(* IEC 61131-3 sources: std_i2980_v2.06_cp053/Source/IMM/ieccontrol/Scope (part 2) *)

(* ---- ABScopeTrigger.pu ---- *)
(*
@h    ! WARNING !
@h    The Kemro K2 system (including software) only meets category B according to EN 954-1,
@h    thus it is not intended for usage in safety-relevant control applications in the field
@h    of personal safety (e.g. emergency stop).
@h    To implement potentially necessary safety-relevant control tasks, always use additional
@h    external safety devices that are intended for the particular purpose, and meet the necessary
@h    functional safety.
@h    For further information see EN 954-1 (EN ISO 13849-1) and/or the K2-x00 user manual, chapter
@h    "CE conformity, directives and standards".

*)

IMPORT_OVER_LISTFILE
 START_PROCESS_ALGORITHM
, cCompMold
, cMoveFwdInterPos
, cMoveFwd
, cMoveBwd
, cMoveBwdInterPos
, cCompInjection
, cMoveInject
, cMovePlast
, TON
, tevMovementState
, tpTriggerData
, tsTriggerData
, tevMovementStateData
, tnActiveInactive

END_IMPORT

ALGORITHM_BLOCK ABScopeTrigger #DUMMY_EDIT_BLOCK

SYSTEM_OBJECT
 PU_Task_7 : TASK;
 EV_Task_3 : TASK;
 Task10ms : TASK;
 evMovementState : tevMovementState;
END_OBJECT

VAR
 fbTimer : TON;
 mevMovementState : tevMovementState (* movement state event *);
 mpbCustomVarTriggerPU : REFTO BOOL;
 mpTriggerPU : tpTriggerData;
 mpTrigger : tpTriggerData;
 mbInit : BOOL;
END_VAR

ALGORITHM aReset

#BEGIN_EDIT_BLOCK
(**************************************** WARNING ********************************************
 *** The KEBA Kemro K2 System including software is not intended for safety control tasks! ***
 ***                       For further information see Comment tab!                        ***
 *********************************************************************************************)

IF (NOT mbInit) THEN
   RETURN;
END_IF;

mpTrigger^.iState := 0;
mpTrigger^.Reduction.iAct := 0;

;#END_EDIT_BLOCK END_ALGORITHM

FUNCTION fArm : BOOL
 #DUMMY_EDIT_BLOCK

VAR_INPUT
 bArm : BOOL (* true activates the waiting for the trigger event *);
END_VAR
#BEGIN_EDIT_BLOCK
(**************************************** WARNING ********************************************
 *** The KEBA Kemro K2 System including software is not intended for safety control tasks! ***
 ***                       For further information see Comment tab!                        ***
 *********************************************************************************************)

IF (NOT mbInit) THEN
   RETURN;
END_IF;

mpTrigger^.bTriggered := FALSE;
mpTrigger^.bPreTriggered := FALSE;
mevMovementState := EMPTY;
mpbCustomVarTriggerPU := EMPTY;
mpTriggerPU := EMPTY;

STOP_PROCESS_ALGORITHM(paTriggerDelay);

IF bArm THEN
   // activate the events
   CASE mpTrigger^.iTriggerIdx OF
      0: // no trigger
         RETURN;

      1..4: // movement triggers
         mevMovementState := evMovementState;

      5: // variable trigger
         mpTrigger^.pbCustomVarTrigger^ := FALSE;
         mpbCustomVarTriggerPU := mpTrigger^.pbCustomVarTrigger;

   END_CASE;
   mpTriggerPU := mpTrigger;
   mpTrigger^.Reduction.iAct := 0;
   mpTrigger^.iState := 1;
END_IF;

fArm := TRUE;

;#END_EDIT_BLOCK END_FUNCTION

FUNCTION fCheckMovementTrigger : BOOL
 #DUMMY_EDIT_BLOCK

VAR_INPUT
 triggerData : tsTriggerData;
 evMovementStateData : tevMovementStateData;
END_VAR

VAR
 nState : tnActiveInactive;
END_VAR
#BEGIN_EDIT_BLOCK
(**************************************** WARNING ********************************************
 *** The KEBA Kemro K2 System including software is not intended for safety control tasks! ***
 ***                       For further information see Comment tab!                        ***
 *********************************************************************************************)

fCheckMovementTrigger := FALSE;

nState := nActive;
IF (triggerData.bFallingEdge) THEN
   nState := nInactive;
END_IF;

IF (evMovementStateData.State = nState) AND
   (//mold close (interposition)
   (triggerData.iTriggerIdx = 1 AND evMovementStateData.DeviceId.CompId = cCompMold AND
   evMovementStateData.DeviceId.IndexId = 1 AND (evMovementStateData.MoveId = cMoveFwdInterPos OR evMovementStateData.MoveId = cMoveFwd) AND
   evMovementStateData.MoveDir = cMoveFwd) OR
   //mold open (interposition)
   (triggerData.iTriggerIdx = 2 AND evMovementStateData.DeviceId.CompId = cCompMold AND
   evMovementStateData.DeviceId.IndexId = 1 AND (evMovementStateData.MoveId = cMoveBwdInterPos OR evMovementStateData.MoveId = cMoveBwd) AND
   evMovementStateData.MoveDir = cMoveBwd) OR
   //inject
   (triggerData.iTriggerIdx = 3 AND evMovementStateData.DeviceId.CompId = cCompInjection AND
   evMovementStateData.DeviceId.IndexId = 1 AND evMovementStateData.MoveId = cMoveInject AND
   evMovementStateData.MoveDir = cMoveFwd) OR
   //plast
   (triggerData.iTriggerIdx = 4 AND evMovementStateData.DeviceId.CompId = cCompInjection AND
   evMovementStateData.DeviceId.IndexId = 1 AND evMovementStateData.MoveId = cMovePlast AND
   evMovementStateData.MoveDir = cMoveBwd)) THEN

   fCheckMovementTrigger := TRUE;
END_IF;

;#END_EDIT_BLOCK END_FUNCTION

ALGORITHM aTrigger

#BEGIN_EDIT_BLOCK
(**************************************** WARNING ********************************************
 *** The KEBA Kemro K2 System including software is not intended for safety control tasks! ***
 ***                       For further information see Comment tab!                        ***
 *********************************************************************************************)

// after ingnition occured, trigger immediately or wait until delay expired
IF (mpTrigger^.dTriggerDelay > t#0.0s) THEN
   fbTimer(IN := FALSE);
   START_PROCESS_ALGORITHM(paTriggerDelay);
ELSE
   // trigger immediately
   mpTrigger^.bTriggered := TRUE;
   mpTrigger^.iState := 2;
END_IF;

;#END_EDIT_BLOCK END_ALGORITHM

ALGORITHM aInit

VAR_INPUT
 pTrigger : tpTriggerData;
END_VAR

VAR
 b : BOOL;
END_VAR
#BEGIN_EDIT_BLOCK
(**************************************** WARNING ********************************************
 *** The KEBA Kemro K2 System including software is not intended for safety control tasks! ***
 ***                       For further information see Comment tab!                        ***
 *********************************************************************************************)

mpTrigger := pTrigger;
mpTriggerPU := EMPTY;
mpbCustomVarTriggerPU := EMPTY;

fbTimer(IN := FALSE);

b := fArm(FALSE);
aReset();

mbInit := TRUE;

;#END_EDIT_BLOCK END_ALGORITHM

PROCESS_ALGORITHM paTriggerDelay ON Task10ms

#BEGIN_EDIT_BLOCK
(**************************************** WARNING ********************************************
 *** The KEBA Kemro K2 System including software is not intended for safety control tasks! ***
 ***                       For further information see Comment tab!                        ***
 *********************************************************************************************)

fbTimer(IN := TRUE, PT := mpTrigger^.dTriggerDelay);

IF fbTimer.Q THEN
   // time-trigger after trigger is ignited and delay is expired
   mpTrigger^.bTriggered := TRUE;
   mpTrigger^.iState := 2;
   STOP_PROCESS_ALGORITHM();
END_IF;

;#END_EDIT_BLOCK END_ALGORITHM

POSTUPDATE_ALGORITHM pPreTriggered ON PU_Task_7 WITH mpTriggerPU^.bPreTriggered

#BEGIN_EDIT_BLOCK
(**************************************** WARNING ********************************************
 *** The KEBA Kemro K2 System including software is not intended for safety control tasks! ***
 ***                       For further information see Comment tab!                        ***
 *********************************************************************************************)

IF (NOT mbInit) THEN
   RETURN;
END_IF;

IF (mpTrigger^.bPreTriggered AND mpTrigger^.Reduction.iAct < mpTrigger^.Reduction.iSet) THEN

   mpTrigger^.Reduction.iAct := mpTrigger^.Reduction.iAct + 1;
   IF (mpTrigger^.Reduction.iAct = mpTrigger^.Reduction.iSet) THEN
      aTrigger();
   END_IF;
   mpTrigger^.bPreTriggered := FALSE;
END_IF;

;#END_EDIT_BLOCK END_ALGORITHM

POSTUPDATE_ALGORITHM pVarTriggered ON PU_Task_7 WITH mpbCustomVarTriggerPU^

#BEGIN_EDIT_BLOCK
(**************************************** WARNING ********************************************
 *** The KEBA Kemro K2 System including software is not intended for safety control tasks! ***
 ***                       For further information see Comment tab!                        ***
 *********************************************************************************************)

IF (mpTrigger^.iTriggerIdx = 5) THEN
   IF ((mpbCustomVarTriggerPU^ AND NOT mpTrigger^.bFallingEdge) OR
       (NOT mpbCustomVarTriggerPU^ AND mpTrigger^.bFallingEdge)) THEN
      mpTrigger^.bPreTriggered := TRUE;
   END_IF;
END_IF;

;#END_EDIT_BLOCK END_ALGORITHM

EVENT_ALGORITHM evaMovementState ON EV_Task_3 WITH mevMovementState

VAR_INPUT
 evMovementStateData : tevMovementStateData;
END_VAR
#BEGIN_EDIT_BLOCK
(**************************************** WARNING ********************************************
 *** The KEBA Kemro K2 System including software is not intended for safety control tasks! ***
 ***                       For further information see Comment tab!                        ***
 *********************************************************************************************)

IF fCheckMovementTrigger(mpTrigger^, evMovementStateData) THEN
   mpTrigger^.bPreTriggered := TRUE;
END_IF;

;#END_EDIT_BLOCK END_ALGORITHM

END_ALGORITHM_BLOCK

#END_OF_IEC_PART

@Puma @IecEditor 6 150 @Pou 25
@@@BEG_Comment@@@
@h    ! WARNING !
@h    The Kemro K2 system (including software) only meets category B according to EN 954-1,
@h    thus it is not intended for usage in safety-relevant control applications in the field
@h    of personal safety (e.g. emergency stop).
@h    To implement potentially necessary safety-relevant control tasks, always use additional
@h    external safety devices that are intended for the particular purpose, and meet the necessary
@h    functional safety.
@h    For further information see EN 954-1 (EN ISO 13849-1) and/or the K2-x00 user manual, chapter
@h    "CE conformity, directives and standards".

@@@END_Comment@@@

@BEG_Contents

@BEG_Func
@RT(17)FuncTreeContainer
1
@Var @RT(23)START_PROCESS_ALGORITHM @RT(0) @T @T @DERIVED 0 @F @RT(23)KEBA_STANDARD_PROCEDURE @F
@T
@BEG_Attrib
0 @RT(0) @RT(0)
@END_Attrib
1 1 @F @F @F @F

@END_Func

@BEG_Const
@RT(18)ConstTreeContainer
8
@Var @RT(9)cCompMold @RT(0) @T @F @DT @RT(4)DINT @RT(0) @T @T @BASIC 0 @F
@F @F
@T
@BEG_Attrib
0 @RT(3)101 @RT(14)Component Mold
@END_Attrib
1 1 @F @F @F @F

@Var @RT(16)cMoveFwdInterPos @RT(0) @T @F @DT @RT(4)DINT @RT(0) @T @T @BASIC 0 @F
@F @F
@T
@BEG_Attrib
0 @RT(2)17 @RT(37)move forward to intermediate position
@END_Attrib
1 1 @F @F @F @F

@Var @RT(8)cMoveFwd @RT(0) @T @F @DT @RT(4)DINT @RT(0) @T @T @BASIC 0 @F
@F @F
@T
@BEG_Attrib
0 @RT(2)12 @RT(16)movement forward
@END_Attrib
1 1 @F @F @F @F

@Var @RT(8)cMoveBwd @RT(0) @T @F @DT @RT(4)DINT @RT(0) @T @T @BASIC 0 @F
@F @F
@T
@BEG_Attrib
0 @RT(2)11 @RT(17)movement backward
@END_Attrib
1 1 @F @F @F @F

@Var @RT(16)cMoveBwdInterPos @RT(0) @T @F @DT @RT(4)DINT @RT(0) @T @T @BASIC 0 @F
@F @F
@T
@BEG_Attrib
0 @RT(2)16 @RT(38)move backward to intermediate position
@END_Attrib
1 1 @F @F @F @F

@Var @RT(14)cCompInjection @RT(0) @T @F @DT @RT(4)DINT @RT(0) @T @T @BASIC 0 @F
@F @F
@T
@BEG_Attrib
0 @RT(3)104 @RT(19)Component Injection
@END_Attrib
1 1 @F @F @F @F

@Var @RT(11)cMoveInject @RT(0) @T @F @DT @RT(4)DINT @RT(0) @T @T @BASIC 0 @F
@F @F
@T
@BEG_Attrib
0 @RT(2)14 @RT(15)inject movement
@END_Attrib
1 1 @F @F @F @F

@Var @RT(10)cMovePlast @RT(0) @T @F @DT @RT(4)DINT @RT(0) @T @T @BASIC 0 @F
@F @F
@T
@BEG_Attrib
0 @RT(2)13 @RT(23)plast movement (rotate)
@END_Attrib
1 1 @F @F @F @F

@END_Const

@BEG_Export

@BEG_Kind
@ALGORITHM_BLOCK @RT(14)ABScopeTrigger @STRUCTURED_TEXT
@RT(0) @RT(0) @RT(0)
@END_Kind

@BEG_Dcl
@RT(16)DclTreeContainer
10
@Var @RT(9)PU_Task_7 @RT(0) @T @F @DT @RT(4)TASK @RT(0) @T @T @BASIC 0 @F
@F @F
@T
@BEG_Attrib
3 @RT(0) @RT(0) @RT(0)
@END_Attrib
1 7 @F @F @F @F

@Var @RT(9)EV_Task_3 @RT(0) @T @F @DT @RT(4)TASK @RT(0) @T @T @BASIC 0 @F
@F @F
@T
@BEG_Attrib
3 @RT(0) @RT(0) @RT(0)
@END_Attrib
1 7 @F @F @F @F

@Var @RT(8)Task10ms @RT(0) @T @T @RENAMED 0 @T @T @DT @RT(4)TASK @RT(0) @T @T @BASIC 0 @F
@F @F
@T
@BEG_Attrib
3 @RT(0) @RT(0) @RT(0)
@END_Attrib
1 7 @F @F @F @F

@Var @RT(7)fbTimer @RT(0) @T @T @DERIVED 0 @T @T @DT @RT(3)TON @RT(0) @T @T @UNKNOWN 0 @F
@F @F
@T
@BEG_Attrib
3 @RT(0) @RT(0) @RT(0)
@END_Attrib
1 0 @F @F @F @F

@Var @RT(15)evMovementState @RT(0) @T @T @DERIVED 0 @T @T @DT @RT(16)tevMovementState @RT(0) @T @T @UNKNOWN 0 @F
@F @F
@T
@BEG_Attrib
3 @RT(0) @RT(0) @RT(0)
@END_Attrib
1 7 @F @F @F @F

@Var @RT(16)mevMovementState @RT(0) @T @T @DERIVED 0 @T @T @DT @RT(16)tevMovementState @RT(0) @T @T @UNKNOWN 0 @F
@F @F
@T
@BEG_Attrib
3 @RT(0) @RT(20)movement state event @RT(0)
@END_Attrib
1 0 @F @F @F @F

@Var @RT(21)mpbCustomVarTriggerPU @RT(0) @T @T @REFTO 0 @T @DT @RT(4)BOOL @RT(0) @T @T @BASIC 0 @F
@F @F
@T
@BEG_Attrib
3 @RT(0) @RT(0) @RT(0)
@END_Attrib
1 0 @F @F @F @F

@Var @RT(11)mpTriggerPU @RT(0) @T @T @DERIVED 0 @T @T @DT @RT(13)tpTriggerData @RT(0) @T @T @UNKNOWN 0 @F
@F @F
@T
@BEG_Attrib
3 @RT(0) @RT(0) @RT(0)
@END_Attrib
1 0 @F @F @F @F

@Var @RT(9)mpTrigger @RT(0) @T @T @RENAMED 0 @T @T @DT @RT(13)tpTriggerData @RT(0) @T @T @UNKNOWN 0 @F
@F @F
@T
@BEG_Attrib
3 @RT(0) @RT(0) @RT(0)
@END_Attrib
1 0 @F @F @F @F

@Var @RT(6)mbInit @RT(0) @T @F @DT @RT(4)BOOL @RT(0) @T @T @BASIC 0 @F
@F @F
@T
@BEG_Attrib
3 @RT(0) @RT(0) @RT(0)
@END_Attrib
1 0 @F @F @F @F

@END_Dcl

@END_Export

@BEG_Body

9

@BEG_Export

@BEG_Algo
@ALGORITHM @RT(6)aReset @STRUCTURED_TEXT
@RT(0) @RT(0) @RT(0) @F @F
@END_Algo

@BEG_Dcl
@RT(16)DclTreeContainer
0
@END_Dcl

@END_Export

@BEG_Export

@BEG_Algo
@FUNCTION @RT(4)fArm @STRUCTURED_TEXT
@RT(4)BOOL @RT(0) @RT(0) @F @F
@END_Algo

@BEG_Dcl
@RT(16)DclTreeContainer
1
@Var @RT(4)bArm @RT(0) @T @F @DT @RT(4)BOOL @RT(0) @T @T @BASIC 0 @F
@F @F
@T
@BEG_Attrib
3 @RT(0) @RT(48)true activates the waiting for the trigger event @RT(0)
@END_Attrib
1 1 @F @F @F @F

@END_Dcl

@END_Export

@BEG_Export

@BEG_Algo
@FUNCTION @RT(21)fCheckMovementTrigger @STRUCTURED_TEXT
@RT(4)BOOL @RT(0) @RT(0) @F @F
@END_Algo

@BEG_Dcl
@RT(16)DclTreeContainer
3
@Var @RT(11)triggerData @RT(0) @T @T @DERIVED 0 @T @T @DT @RT(13)tsTriggerData @RT(0) @T @T @UNKNOWN 0 @F
@F @F
@T
@BEG_Attrib
3 @RT(0) @RT(0) @RT(0)
@END_Attrib
1 1 @F @F @F @F

@Var @RT(19)evMovementStateData @RT(0) @T @T @DERIVED 0 @T @T @DT @RT(20)tevMovementStateData @RT(0) @T @T @UNKNOWN 0 @F
@F @F
@T
@BEG_Attrib
3 @RT(0) @RT(0) @RT(0)
@END_Attrib
1 1 @F @F @F @F

@Var @RT(6)nState @RT(0) @T @T @DERIVED 0 @T @T @DT @RT(16)tnActiveInactive @RT(0) @T @T @UNKNOWN 0 @F
@F @F
@T
@BEG_Attrib
3 @RT(0) @RT(0) @RT(0)
@END_Attrib
1 0 @F @F @F @F

@END_Dcl

@END_Export

@BEG_Export

@BEG_Algo
@ALGORITHM @RT(8)aTrigger @STRUCTURED_TEXT
@RT(0) @RT(0) @RT(0) @F @F
@END_Algo

@BEG_Dcl
@RT(16)DclTreeContainer
0
@END_Dcl

@END_Export

@BEG_Export

@BEG_Algo
@ALGORITHM @RT(5)aInit @STRUCTURED_TEXT
@RT(0) @RT(0) @RT(0) @F @F
@END_Algo

@BEG_Dcl
@RT(16)DclTreeContainer
2
@Var @RT(8)pTrigger @RT(0) @T @T @DERIVED 0 @T @T @DT @RT(13)tpTriggerData @RT(0) @T @T @UNKNOWN 0 @F
@F @F
@T
@BEG_Attrib
3 @RT(0) @RT(0) @RT(0)
@END_Attrib
1 1 @F @F @F @F

@Var @RT(1)b @RT(0) @T @F @DT @RT(4)BOOL @RT(0) @T @T @BASIC 0 @F
@F @F
@T
@BEG_Attrib
3 @RT(0) @RT(0) @RT(0)
@END_Attrib
1 0 @F @F @F @F

@END_Dcl

@END_Export

@BEG_Export

@BEG_Algo
@PROCESS_ALGORITHM @RT(14)paTriggerDelay @STRUCTURED_TEXT
@RT(0) @RT(0) @RT(8)Task10ms @F @F
@END_Algo

@BEG_Dcl
@RT(16)DclTreeContainer
0
@END_Dcl

@END_Export

@BEG_Export

@BEG_Algo
@POSTUPDATE_ALGORITHM @RT(13)pPreTriggered @STRUCTURED_TEXT
@RT(0) @RT(26)mpTriggerPU^.bPreTriggered @RT(9)PU_Task_7 @F @F
@END_Algo

@BEG_Dcl
@RT(16)DclTreeContainer
0
@END_Dcl

@END_Export

@BEG_Export

@BEG_Algo
@POSTUPDATE_ALGORITHM @RT(13)pVarTriggered @STRUCTURED_TEXT
@RT(0) @RT(22)mpbCustomVarTriggerPU^ @RT(9)PU_Task_7 @F @F
@END_Algo

@BEG_Dcl
@RT(16)DclTreeContainer
0
@END_Dcl

@END_Export

@BEG_Export

@BEG_Algo
@EVENT_ALGORITHM @RT(16)evaMovementState @STRUCTURED_TEXT
@RT(0) @RT(16)mevMovementState @RT(9)EV_Task_3 @F @F
@END_Algo

@BEG_Dcl
@RT(16)DclTreeContainer
1
@Var @RT(19)evMovementStateData @RT(0) @T @T @DERIVED 0 @T @T @DT @RT(20)tevMovementStateData @RT(0) @T @T @UNKNOWN 0 @F
@F @F
@T
@BEG_Attrib
3 @RT(0) @RT(0) @RT(0)
@END_Attrib
1 1 @F @F @F @F

@END_Dcl

@END_Export

@BEG_Body
@TL(14)
(**************************************** WARNING ********************************************
 *** The KEBA Kemro K2 System including software is not intended for safety control tasks! ***
 ***                       For further information see Comment tab!                        ***
 *********************************************************************************************)

IF (NOT mbInit) THEN
   RETURN;
END_IF;

mpTrigger^.iState := 0;
mpTrigger^.Reduction.iAct := 0;

@END_Body

@@@BEG_Comment@@@
@TL(0)

@@@END_Comment@@@

@BEG_Body
@TL(40)
(**************************************** WARNING ********************************************
 *** The KEBA Kemro K2 System including software is not intended for safety control tasks! ***
 ***                       For further information see Comment tab!                        ***
 *********************************************************************************************)

IF (NOT mbInit) THEN
   RETURN;
END_IF;

mpTrigger^.bTriggered := FALSE;
mpTrigger^.bPreTriggered := FALSE;
mevMovementState := EMPTY;
mpbCustomVarTriggerPU := EMPTY;
mpTriggerPU := EMPTY;

STOP_PROCESS_ALGORITHM(paTriggerDelay);

IF bArm THEN
   // activate the events
   CASE mpTrigger^.iTriggerIdx OF
      0: // no trigger
         RETURN;

      1..4: // movement triggers
         mevMovementState := evMovementState;

      5: // variable trigger
         mpTrigger^.pbCustomVarTrigger^ := FALSE;
         mpbCustomVarTriggerPU := mpTrigger^.pbCustomVarTrigger;

   END_CASE;
   mpTriggerPU := mpTrigger;
   mpTrigger^.Reduction.iAct := 0;
   mpTrigger^.iState := 1;
END_IF;

fArm := TRUE;

@END_Body

@@@BEG_Comment@@@
@TL(0)

@@@END_Comment@@@

@BEG_Body
@TL(36)
(**************************************** WARNING ********************************************
 *** The KEBA Kemro K2 System including software is not intended for safety control tasks! ***
 ***                       For further information see Comment tab!                        ***
 *********************************************************************************************)

fCheckMovementTrigger := FALSE;

nState := nActive;
IF (triggerData.bFallingEdge) THEN
   nState := nInactive;
END_IF;

IF (evMovementStateData.State = nState) AND
   (//mold close (interposition)
   (triggerData.iTriggerIdx = 1 AND evMovementStateData.DeviceId.CompId = cCompMold AND
   evMovementStateData.DeviceId.IndexId = 1 AND (evMovementStateData.MoveId = cMoveFwdInterPos OR evMovementStateData.MoveId = cMoveFwd) AND
   evMovementStateData.MoveDir = cMoveFwd) OR
   //mold open (interposition)
   (triggerData.iTriggerIdx = 2 AND evMovementStateData.DeviceId.CompId = cCompMold AND
   evMovementStateData.DeviceId.IndexId = 1 AND (evMovementStateData.MoveId = cMoveBwdInterPos OR evMovementStateData.MoveId = cMoveBwd) AND
   evMovementStateData.MoveDir = cMoveBwd) OR
   //inject
   (triggerData.iTriggerIdx = 3 AND evMovementStateData.DeviceId.CompId = cCompInjection AND
   evMovementStateData.DeviceId.IndexId = 1 AND evMovementStateData.MoveId = cMoveInject AND
   evMovementStateData.MoveDir = cMoveFwd) OR
   //plast
   (triggerData.iTriggerIdx = 4 AND evMovementStateData.DeviceId.CompId = cCompInjection AND
   evMovementStateData.DeviceId.IndexId = 1 AND evMovementStateData.MoveId = cMovePlast AND
   evMovementStateData.MoveDir = cMoveBwd)) THEN

   fCheckMovementTrigger := TRUE;
END_IF;

@END_Body

@@@BEG_Comment@@@
@TL(0)

@@@END_Comment@@@

@BEG_Body
@TL(15)
(**************************************** WARNING ********************************************
 *** The KEBA Kemro K2 System including software is not intended for safety control tasks! ***
 ***                       For further information see Comment tab!                        ***
 *********************************************************************************************)

// after ingnition occured, trigger immediately or wait until delay expired
IF (mpTrigger^.dTriggerDelay > t#0.0s) THEN
   fbTimer(IN := FALSE);
   START_PROCESS_ALGORITHM(paTriggerDelay);
ELSE
   // trigger immediately
   mpTrigger^.bTriggered := TRUE;
   mpTrigger^.iState := 2;
END_IF;

@END_Body

@@@BEG_Comment@@@
@TL(0)

@@@END_Comment@@@

@BEG_Body
@TL(16)
(**************************************** WARNING ********************************************
 *** The KEBA Kemro K2 System including software is not intended for safety control tasks! ***
 ***                       For further information see Comment tab!                        ***
 *********************************************************************************************)

mpTrigger := pTrigger;
mpTriggerPU := EMPTY;
mpbCustomVarTriggerPU := EMPTY;

fbTimer(IN := FALSE);

b := fArm(FALSE);
aReset();

mbInit := TRUE;

@END_Body

@@@BEG_Comment@@@
@TL(0)

@@@END_Comment@@@

@BEG_Body
@TL(14)
(**************************************** WARNING ********************************************
 *** The KEBA Kemro K2 System including software is not intended for safety control tasks! ***
 ***                       For further information see Comment tab!                        ***
 *********************************************************************************************)

fbTimer(IN := TRUE, PT := mpTrigger^.dTriggerDelay);

IF fbTimer.Q THEN
   // time-trigger after trigger is ignited and delay is expired
   mpTrigger^.bTriggered := TRUE;
   mpTrigger^.iState := 2;
   STOP_PROCESS_ALGORITHM();
END_IF;

@END_Body

@@@BEG_Comment@@@
@TL(0)

@@@END_Comment@@@

@BEG_Body
@TL(22)
(**************************************** WARNING ********************************************
 *** The KEBA Kemro K2 System including software is not intended for safety control tasks! ***
 ***                       For further information see Comment tab!                        ***
 *********************************************************************************************)

IF (NOT mbInit) THEN
   RETURN;
END_IF;

IF (mpTrigger^.bPreTriggered AND mpTrigger^.Reduction.iAct < mpTrigger^.Reduction.iSet) THEN

   mpTrigger^.Reduction.iAct := mpTrigger^.Reduction.iAct + 1;
   IF (mpTrigger^.Reduction.iAct = mpTrigger^.Reduction.iSet) THEN
      aTrigger();
   END_IF;
   mpTrigger^.bPreTriggered := FALSE;
END_IF;

@END_Body

@@@BEG_Comment@@@
@TL(0)

@@@END_Comment@@@

@BEG_Body
@TL(12)
(**************************************** WARNING ********************************************
 *** The KEBA Kemro K2 System including software is not intended for safety control tasks! ***
 ***                       For further information see Comment tab!                        ***
 *********************************************************************************************)

IF (mpTrigger^.iTriggerIdx = 5) THEN
   IF ((mpbCustomVarTriggerPU^ AND NOT mpTrigger^.bFallingEdge) OR
       (NOT mpbCustomVarTriggerPU^ AND mpTrigger^.bFallingEdge)) THEN
      mpTrigger^.bPreTriggered := TRUE;
   END_IF;
END_IF;

@END_Body

@@@BEG_Comment@@@
@TL(0)

@@@END_Comment@@@

@BEG_Body
@TL(10)
(**************************************** WARNING ********************************************
 *** The KEBA Kemro K2 System including software is not intended for safety control tasks! ***
 ***                       For further information see Comment tab!                        ***
 *********************************************************************************************)

IF fCheckMovementTrigger(mpTrigger^, evMovementStateData) THEN
   mpTrigger^.bPreTriggered := TRUE;
END_IF;

@END_Body

@@@BEG_Comment@@@
@TL(0)

@@@END_Comment@@@
@END_Body

@END_Contents

(* ---- FAddVarToScope.pu ---- *)
(*
@h    ! WARNING !
@h    The Kemro K2 system (including software) only meets category B according to EN 954-1,
@h    thus it is not intended for usage in safety-relevant control applications in the field
@h    of personal safety (e.g. emergency stop).
@h    To implement potentially necessary safety-relevant control tasks, always use additional
@h    external safety devices that are intended for the particular purpose, and meet the necessary
@h    functional safety.
@h    For further information see EN 954-1 (EN ISO 13849-1) and/or the K2-x00 user manual, chapter
@h    "CE conformity, directives and standards".

*)

IMPORT_OVER_LISTFILE
 tnSVDataTypes
, tsSV
//  tsScopeVar
, KSWO_Status

END_IMPORT

FUNCTION FAddVarToScope : BOOL #DUMMY_EDIT_BLOCK

VAR_INPUT
 Name : STRING(255);
 Task : TASK;
 SysVarType : tnSVDataTypes;
END_VAR

VAR_IN_OUT
 SysVar : tsSV;
 // scopeVar : tsScopeVar;
END_VAR

VAR
 swoState : KSWO_Status;
END_VAR
#BEGIN_EDIT_BLOCK
(**************************************** WARNING ********************************************
 *** The KEBA Kemro K2 System including software is not intended for safety control tasks! ***
 ***                       For further information see Comment tab!                        ***
 *********************************************************************************************)

CASE SysVarType OF
   nDT_BOOL  : swoState := KSWO_AddVariable(Task := Task, Name := Name, Variable := SysVar.pbBOOLSV^);
   nDT_BYTE  : swoState := KSWO_AddVariable(Task := Task, Name := Name, Variable := SysVar.piBYTESV^);
   nDT_WORD  : swoState := KSWO_AddVariable(Task := Task, Name := Name, Variable := SysVar.piWORDSV^);
   nDT_DWORD : swoState := KSWO_AddVariable(Task := Task, Name := Name, Variable := SysVar.piDWORDSV^);
   nDT_LWORD : swoState := KSWO_AddVariable(Task := Task, Name := Name, Variable := SysVar.piLWORDSV^);
   nDT_INT   : swoState := KSWO_AddVariable(Task := Task, Name := Name, Variable := SysVar.piINTSV^);
   nDT_UINT  : swoState := KSWO_AddVariable(Task := Task, Name := Name, Variable := SysVar.piUINTSV^);
   nDT_DINT  : swoState := KSWO_AddVariable(Task := Task, Name := Name, Variable := SysVar.piDINTSV^);
   nDT_UDINT : swoState := KSWO_AddVariable(Task := Task, Name := Name, Variable := SysVar.piUDINTSV^);
   nDT_SINT  : swoState := KSWO_AddVariable(Task := Task, Name := Name, Variable := SysVar.piSINTSV^);
   nDT_USINT : swoState := KSWO_AddVariable(Task := Task, Name := Name, Variable := SysVar.piUSINTSV^);
   nDT_LINT  : swoState := KSWO_AddVariable(Task := Task, Name := Name, Variable := SysVar.piLINTSV^);
   nDT_ULINT : swoState := KSWO_AddVariable(Task := Task, Name := Name, Variable := SysVar.piULINTSV^);
   nDT_REAL  : swoState := KSWO_AddVariable(Task := Task, Name := Name, Variable := SysVar.prREALSV^);
   nDT_LREAL : swoState := KSWO_AddVariable(Task := Task, Name := Name, Variable := SysVar.prLREALSV^);
   nDT_TIME  : swoState := KSWO_AddVariable(Task := Task, Name := Name, Variable := SysVar.pdTIMESV^);
ELSE
   FAddVarToScope := FALSE;
   RETURN;
END_CASE;

FAddVarToScope := (swoState <> KSWO_Status_OK);

;#END_EDIT_BLOCK END_FUNCTION

#END_OF_IEC_PART

@Puma @IecEditor 6 150 @Pou 25
@@@BEG_Comment@@@
@h    ! WARNING !
@h    The Kemro K2 system (including software) only meets category B according to EN 954-1,
@h    thus it is not intended for usage in safety-relevant control applications in the field
@h    of personal safety (e.g. emergency stop).
@h    To implement potentially necessary safety-relevant control tasks, always use additional
@h    external safety devices that are intended for the particular purpose, and meet the necessary
@h    functional safety.
@h    For further information see EN 954-1 (EN ISO 13849-1) and/or the K2-x00 user manual, chapter
@h    "CE conformity, directives and standards".

@@@END_Comment@@@

@BEG_Contents

@BEG_Func
@RT(17)FuncTreeContainer
0
@END_Func

@BEG_Const
@RT(18)ConstTreeContainer
0
@END_Const

@BEG_Export

@BEG_Kind
@FUNCTION @RT(14)FAddVarToScope @STRUCTURED_TEXT
@RT(4)BOOL @RT(0) @RT(0)
@END_Kind

@BEG_Dcl
@RT(16)DclTreeContainer
6
@Var @RT(4)Name @RT(0) @T @F @DT @RT(11)STRING(255) @RT(0) @T @T @STRING 0 @F @RT(3)255 @F
@F @F
@T
@BEG_Attrib
3 @RT(0) @RT(0) @RT(0)
@END_Attrib
1 1 @F @F @F @F

@Var @RT(4)Task @RT(0) @T @F @DT @RT(4)TASK @RT(0) @T @T @BASIC 0 @F
@F @F
@T
@BEG_Attrib
3 @RT(0) @RT(0) @RT(0)
@END_Attrib
1 1 @F @F @F @F

@Var @RT(10)SysVarType @RT(0) @T @T @DERIVED 0 @T @T @DT @RT(13)tnSVDataTypes @RT(0) @T @T @UNKNOWN 0 @F
@F @F
@T
@BEG_Attrib
3 @RT(0) @RT(0) @RT(0)
@END_Attrib
1 1 @F @F @F @F

@Var @RT(6)SysVar @RT(0) @T @T @DERIVED 0 @T @T @DT @RT(4)tsSV @RT(0) @T @T @UNKNOWN 0 @F
@F @F
@T
@BEG_Attrib
3 @RT(0) @RT(0) @RT(0)
@END_Attrib
1 2 @F @F @F @F

@Var @RT(8)scopeVar @RT(0) @T @T @DERIVED 0 @T @T @DT @RT(10)tsScopeVar @RT(0) @T @T @UNKNOWN 0 @F
@F @T
@T
@BEG_Attrib
3 @RT(0) @RT(0) @RT(0)
@END_Attrib
1 2 @F @F @F @F

@Var @RT(8)swoState @RT(0) @T @T @DERIVED 0 @T @T @DT @RT(11)KSWO_Status @RT(0) @T @T @UNKNOWN 0 @F
@F @F
@T
@BEG_Attrib
3 @RT(0) @RT(0) @RT(0)
@END_Attrib
1 0 @F @F @F @F

@END_Dcl

@END_Export

@BEG_Body
@TL(31)
(**************************************** WARNING ********************************************
 *** The KEBA Kemro K2 System including software is not intended for safety control tasks! ***
 ***                       For further information see Comment tab!                        ***
 *********************************************************************************************)

CASE SysVarType OF
   nDT_BOOL  : swoState := KSWO_AddVariable(Task := Task, Name := Name, Variable := SysVar.pbBOOLSV^);
   nDT_BYTE  : swoState := KSWO_AddVariable(Task := Task, Name := Name, Variable := SysVar.piBYTESV^);
   nDT_WORD  : swoState := KSWO_AddVariable(Task := Task, Name := Name, Variable := SysVar.piWORDSV^);
   nDT_DWORD : swoState := KSWO_AddVariable(Task := Task, Name := Name, Variable := SysVar.piDWORDSV^);
   nDT_LWORD : swoState := KSWO_AddVariable(Task := Task, Name := Name, Variable := SysVar.piLWORDSV^);
   nDT_INT   : swoState := KSWO_AddVariable(Task := Task, Name := Name, Variable := SysVar.piINTSV^);
   nDT_UINT  : swoState := KSWO_AddVariable(Task := Task, Name := Name, Variable := SysVar.piUINTSV^);
   nDT_DINT  : swoState := KSWO_AddVariable(Task := Task, Name := Name, Variable := SysVar.piDINTSV^);
   nDT_UDINT : swoState := KSWO_AddVariable(Task := Task, Name := Name, Variable := SysVar.piUDINTSV^);
   nDT_SINT  : swoState := KSWO_AddVariable(Task := Task, Name := Name, Variable := SysVar.piSINTSV^);
   nDT_USINT : swoState := KSWO_AddVariable(Task := Task, Name := Name, Variable := SysVar.piUSINTSV^);
   nDT_LINT  : swoState := KSWO_AddVariable(Task := Task, Name := Name, Variable := SysVar.piLINTSV^);
   nDT_ULINT : swoState := KSWO_AddVariable(Task := Task, Name := Name, Variable := SysVar.piULINTSV^);
   nDT_REAL  : swoState := KSWO_AddVariable(Task := Task, Name := Name, Variable := SysVar.prREALSV^);
   nDT_LREAL : swoState := KSWO_AddVariable(Task := Task, Name := Name, Variable := SysVar.prLREALSV^);
   nDT_TIME  : swoState := KSWO_AddVariable(Task := Task, Name := Name, Variable := SysVar.pdTIMESV^);
ELSE
   FAddVarToScope := FALSE;
   RETURN;
END_CASE;

FAddVarToScope := (swoState <> KSWO_Status_OK);

@END_Body

@END_Contents

(* ---- FGetSysVarFromName.pu ---- *)
(*
@h    ! WARNING !
@h    The Kemro K2 system (including software) only meets category B according to EN 954-1,
@h    thus it is not intended for usage in safety-relevant control applications in the field
@h    of personal safety (e.g. emergency stop).
@h    To implement potentially necessary safety-relevant control tasks, always use additional
@h    external safety devices that are intended for the particular purpose, and meet the necessary
@h    functional safety.
@h    For further information see EN 954-1 (EN ISO 13849-1) and/or the K2-x00 user manual, chapter
@h    "CE conformity, directives and standards".

*)

IMPORT_OVER_LISTFILE
 tnSVDataTypes
, tsSV
, KSYS_Status

END_IMPORT

FUNCTION FGetSysVarFromName : tnSVDataTypes #DUMMY_EDIT_BLOCK

VAR_INPUT
 Name : STRING(255);
END_VAR

VAR_IN_OUT
 SysVar : tsSV;
END_VAR

VAR
 SysVarTemp : tsSV;
 sysStatus : KSYS_Status;
END_VAR
#BEGIN_EDIT_BLOCK
(**************************************** WARNING ********************************************
 *** The KEBA Kemro K2 System including software is not intended for safety control tasks! ***
 ***                       For further information see Comment tab!                        ***
 *********************************************************************************************)

FGetSysVarFromName := nDT_NONE;

SysVarTemp.prREALSV := GET_SYNC_REFTO(Name, t#0s, sysStatus);
IF sysStatus = KSYS_Status_OK THEN
   SysVar := SysVarTemp;
   FGetSysVarFromName := nDT_REAL;
   RETURN;
END_IF;

SysVarTemp.pbBOOLSV := GET_SYNC_REFTO(Name, t#0s, sysStatus);
IF sysStatus = KSYS_Status_OK THEN
   SysVar := SysVarTemp;
   FGetSysVarFromName := nDT_BOOL;
   RETURN;
END_IF;

SysVarTemp.pdTIMESV := GET_SYNC_REFTO(Name, t#0s, sysStatus);
IF sysStatus = KSYS_Status_OK THEN
   SysVar := SysVarTemp;
   FGetSysVarFromName := nDT_TIME;
   RETURN;
END_IF;

SysVarTemp.piBYTESV := GET_SYNC_REFTO(Name, t#0s, sysStatus);
IF sysStatus = KSYS_Status_OK THEN
   SysVar := SysVarTemp;
   FGetSysVarFromName := nDT_BYTE;
   RETURN;
END_IF;

SysVarTemp.piWORDSV := GET_SYNC_REFTO(Name, t#0s, sysStatus);
IF sysStatus = KSYS_Status_OK THEN
   SysVar := SysVarTemp;
   FGetSysVarFromName := nDT_WORD;
   RETURN;
END_IF;

SysVarTemp.piDWORDSV := GET_SYNC_REFTO(Name, t#0s, sysStatus);
IF sysStatus = KSYS_Status_OK THEN
   SysVar := SysVarTemp;
   FGetSysVarFromName := nDT_DWORD;
   RETURN;
END_IF;

SysVarTemp.piLWORDSV := GET_SYNC_REFTO(Name, t#0s, sysStatus);
IF sysStatus = KSYS_Status_OK THEN
   SysVar := SysVarTemp;
   FGetSysVarFromName := nDT_LWORD;
   RETURN;
END_IF;

SysVarTemp.piINTSV := GET_SYNC_REFTO(Name, t#0s, sysStatus);
IF sysStatus = KSYS_Status_OK THEN
   SysVar := SysVarTemp;
   FGetSysVarFromName := nDT_INT;
   RETURN;
END_IF;

SysVarTemp.piUINTSV := GET_SYNC_REFTO(Name, t#0s, sysStatus);
IF sysStatus = KSYS_Status_OK THEN
   SysVar := SysVarTemp;
   FGetSysVarFromName := nDT_UINT;
   RETURN;
END_IF;

SysVarTemp.piDINTSV := GET_SYNC_REFTO(Name, t#0s, sysStatus);
IF sysStatus = KSYS_Status_OK THEN
   SysVar := SysVarTemp;
   FGetSysVarFromName := nDT_DINT;
   RETURN;
END_IF;

SysVarTemp.piUDINTSV := GET_SYNC_REFTO(Name, t#0s, sysStatus);
IF sysStatus = KSYS_Status_OK THEN
   SysVar := SysVarTemp;
   FGetSysVarFromName := nDT_UDINT;
   RETURN;
END_IF;

SysVarTemp.piSINTSV := GET_SYNC_REFTO(Name, t#0s, sysStatus);
IF sysStatus = KSYS_Status_OK THEN
   SysVar := SysVarTemp;
   FGetSysVarFromName := nDT_SINT;
   RETURN;
END_IF;

SysVarTemp.piUSINTSV := GET_SYNC_REFTO(Name, t#0s, sysStatus);
IF sysStatus = KSYS_Status_OK THEN
   SysVar := SysVarTemp;
   FGetSysVarFromName := nDT_USINT;
   RETURN;
END_IF;

SysVarTemp.piLINTSV := GET_SYNC_REFTO(Name, t#0s, sysStatus);
IF sysStatus = KSYS_Status_OK THEN
   SysVar := SysVarTemp;
   FGetSysVarFromName := nDT_LINT;
   RETURN;
END_IF;

SysVarTemp.piULINTSV := GET_SYNC_REFTO(Name, t#0s, sysStatus);
IF sysStatus = KSYS_Status_OK THEN
   SysVar := SysVarTemp;
   FGetSysVarFromName := nDT_ULINT;
   RETURN;
END_IF;

SysVarTemp.prLREALSV := GET_SYNC_REFTO(Name, t#0s, sysStatus);
IF sysStatus = KSYS_Status_OK THEN
   SysVar := SysVarTemp;
   FGetSysVarFromName := nDT_LREAL;
   RETURN;
END_IF;

;#END_EDIT_BLOCK END_FUNCTION

#END_OF_IEC_PART

@Puma @IecEditor 6 150 @Pou 25
@@@BEG_Comment@@@
@h    ! WARNING !
@h    The Kemro K2 system (including software) only meets category B according to EN 954-1,
@h    thus it is not intended for usage in safety-relevant control applications in the field
@h    of personal safety (e.g. emergency stop).
@h    To implement potentially necessary safety-relevant control tasks, always use additional
@h    external safety devices that are intended for the particular purpose, and meet the necessary
@h    functional safety.
@h    For further information see EN 954-1 (EN ISO 13849-1) and/or the K2-x00 user manual, chapter
@h    "CE conformity, directives and standards".

@@@END_Comment@@@

@BEG_Contents

@BEG_Func
@RT(17)FuncTreeContainer
0
@END_Func

@BEG_Const
@RT(18)ConstTreeContainer
0
@END_Const

@BEG_Export

@BEG_Kind
@FUNCTION @RT(18)FGetSysVarFromName @STRUCTURED_TEXT
@RT(13)tnSVDataTypes @RT(0) @RT(0)
@END_Kind

@BEG_Dcl
@RT(16)DclTreeContainer
4
@Var @RT(4)Name @RT(0) @T @F @DT @RT(11)STRING(255) @RT(0) @T @T @STRING 0 @F @RT(3)255 @F
@F @F
@T
@BEG_Attrib
3 @RT(0) @RT(0) @RT(0)
@END_Attrib
1 1 @F @F @F @F

@Var @RT(6)SysVar @RT(0) @T @T @DERIVED 0 @T @T @DT @RT(4)tsSV @RT(0) @T @T @UNKNOWN 0 @F
@F @F
@T
@BEG_Attrib
3 @RT(0) @RT(0) @RT(0)
@END_Attrib
1 2 @F @F @F @F

@Var @RT(10)SysVarTemp @RT(0) @T @T @DERIVED 0 @T @T @DT @RT(4)tsSV @RT(0) @T @T @UNKNOWN 0 @F
@F @F
@T
@BEG_Attrib
3 @RT(0) @RT(0) @RT(0)
@END_Attrib
1 0 @F @F @F @F

@Var @RT(9)sysStatus @RT(0) @T @T @DERIVED 0 @T @T @DT @RT(11)KSYS_Status @RT(0) @T @T @UNKNOWN 0 @F
@F @F
@T
@BEG_Attrib
3 @RT(0) @RT(0) @RT(0)
@END_Attrib
1 0 @F @F @F @F

@END_Dcl

@END_Export

@BEG_Body
@TL(119)
(**************************************** WARNING ********************************************
 *** The KEBA Kemro K2 System including software is not intended for safety control tasks! ***
 ***                       For further information see Comment tab!                        ***
 *********************************************************************************************)

FGetSysVarFromName := nDT_NONE;

SysVarTemp.prREALSV := GET_SYNC_REFTO(Name, t#0s, sysStatus);
IF sysStatus = KSYS_Status_OK THEN
   SysVar := SysVarTemp;
   FGetSysVarFromName := nDT_REAL;
   RETURN;
END_IF;

SysVarTemp.pbBOOLSV := GET_SYNC_REFTO(Name, t#0s, sysStatus);
IF sysStatus = KSYS_Status_OK THEN
   SysVar := SysVarTemp;
   FGetSysVarFromName := nDT_BOOL;
   RETURN;
END_IF;

SysVarTemp.pdTIMESV := GET_SYNC_REFTO(Name, t#0s, sysStatus);
IF sysStatus = KSYS_Status_OK THEN
   SysVar := SysVarTemp;
   FGetSysVarFromName := nDT_TIME;
   RETURN;
END_IF;

SysVarTemp.piBYTESV := GET_SYNC_REFTO(Name, t#0s, sysStatus);
IF sysStatus = KSYS_Status_OK THEN
   SysVar := SysVarTemp;
   FGetSysVarFromName := nDT_BYTE;
   RETURN;
END_IF;

SysVarTemp.piWORDSV := GET_SYNC_REFTO(Name, t#0s, sysStatus);
IF sysStatus = KSYS_Status_OK THEN
   SysVar := SysVarTemp;
   FGetSysVarFromName := nDT_WORD;
   RETURN;
END_IF;

SysVarTemp.piDWORDSV := GET_SYNC_REFTO(Name, t#0s, sysStatus);
IF sysStatus = KSYS_Status_OK THEN
   SysVar := SysVarTemp;
   FGetSysVarFromName := nDT_DWORD;
   RETURN;
END_IF;

SysVarTemp.piLWORDSV := GET_SYNC_REFTO(Name, t#0s, sysStatus);
IF sysStatus = KSYS_Status_OK THEN
   SysVar := SysVarTemp;
   FGetSysVarFromName := nDT_LWORD;
   RETURN;
END_IF;

SysVarTemp.piINTSV := GET_SYNC_REFTO(Name, t#0s, sysStatus);
IF sysStatus = KSYS_Status_OK THEN
   SysVar := SysVarTemp;
   FGetSysVarFromName := nDT_INT;
   RETURN;
END_IF;

SysVarTemp.piUINTSV := GET_SYNC_REFTO(Name, t#0s, sysStatus);
IF sysStatus = KSYS_Status_OK THEN
   SysVar := SysVarTemp;
   FGetSysVarFromName := nDT_UINT;
   RETURN;
END_IF;

SysVarTemp.piDINTSV := GET_SYNC_REFTO(Name, t#0s, sysStatus);
IF sysStatus = KSYS_Status_OK THEN
   SysVar := SysVarTemp;
   FGetSysVarFromName := nDT_DINT;
   RETURN;
END_IF;

SysVarTemp.piUDINTSV := GET_SYNC_REFTO(Name, t#0s, sysStatus);
IF sysStatus = KSYS_Status_OK THEN
   SysVar := SysVarTemp;
   FGetSysVarFromName := nDT_UDINT;
   RETURN;
END_IF;

SysVarTemp.piSINTSV := GET_SYNC_REFTO(Name, t#0s, sysStatus);
IF sysStatus = KSYS_Status_OK THEN
   SysVar := SysVarTemp;
   FGetSysVarFromName := nDT_SINT;
   RETURN;
END_IF;

SysVarTemp.piUSINTSV := GET_SYNC_REFTO(Name, t#0s, sysStatus);
IF sysStatus = KSYS_Status_OK THEN
   SysVar := SysVarTemp;
   FGetSysVarFromName := nDT_USINT;
   RETURN;
END_IF;

SysVarTemp.piLINTSV := GET_SYNC_REFTO(Name, t#0s, sysStatus);
IF sysStatus = KSYS_Status_OK THEN
   SysVar := SysVarTemp;
   FGetSysVarFromName := nDT_LINT;
   RETURN;
END_IF;

SysVarTemp.piULINTSV := GET_SYNC_REFTO(Name, t#0s, sysStatus);
IF sysStatus = KSYS_Status_OK THEN
   SysVar := SysVarTemp;
   FGetSysVarFromName := nDT_ULINT;
   RETURN;
END_IF;

SysVarTemp.prLREALSV := GET_SYNC_REFTO(Name, t#0s, sysStatus);
IF sysStatus = KSYS_Status_OK THEN
   SysVar := SysVarTemp;
   FGetSysVarFromName := nDT_LREAL;
   RETURN;
END_IF;

@END_Body

@END_Contents

(* ---- FBTimeStamp.pu ---- *)
IMPORT_OVER_LISTFILE
 RTC

END_IMPORT

FUNCTION_BLOCK FBTimeStamp #DUMMY_EDIT_BLOCK

VAR_OUTPUT
 sTimeStamp : STRING(255);
END_VAR

VAR
 fbRTC : RTC;
 sTime : STRING(255);
END_VAR
#BEGIN_EDIT_BLOCK

(**************************************** WARNING ********************************************
 *** The KEBA Kemro K2 System including software is not intended for safety control tasks! ***
 ***                       For further information see Comment tab!                        ***
 *********************************************************************************************)
fbRTC(EN := FALSE);
sTime := DATE_AND_TIME_TO_STRING(fbRTC.CDT); //e.g. DT#2015-08-18-12:03:15.970149
sTimeStamp := CONCAT(MID(sTime, 10,4), '_', MID(sTime, 2, 15), '-',  MID(sTime, 2, 18), '-', MID(sTime, 2, 21)); //yyyy-mm-dd_hh-mm-ss

;#END_EDIT_BLOCK END_FUNCTION_BLOCK

#END_OF_IEC_PART

@Puma @IecEditor 6 150 @Pou 25
@@@BEG_Comment@@@

@@@END_Comment@@@

@BEG_Contents

@BEG_Func
@RT(17)FuncTreeContainer
0
@END_Func

@BEG_Const
@RT(18)ConstTreeContainer
0
@END_Const

@BEG_Export

@BEG_Kind
@FUNCTION_BLOCK @RT(11)FBTimeStamp @STRUCTURED_TEXT
@RT(0) @RT(0) @RT(0)
@END_Kind

@BEG_Dcl
@RT(16)DclTreeContainer
3
@Var @RT(5)fbRTC @RT(0) @T @T @DERIVED 0 @T @T @DT @RT(3)RTC @RT(0) @T @T @UNKNOWN 0 @F
@F @F
@T
@BEG_Attrib
3 @RT(0) @RT(0) @RT(0)
@END_Attrib
1 0 @F @F @F @F

@Var @RT(5)sTime @RT(0) @T @F @DT @RT(11)STRING(255) @RT(0) @T @T @STRING 0 @F @RT(3)255 @F
@F @F
@T
@BEG_Attrib
3 @RT(0) @RT(0) @RT(0)
@END_Attrib
1 0 @F @F @F @F

@Var @RT(10)sTimeStamp @RT(0) @T @F @DT @RT(11)STRING(255) @RT(0) @T @T @STRING 0 @F @RT(3)255 @F
@F @F
@T
@BEG_Attrib
3 @RT(0) @RT(0) @RT(0)
@END_Attrib
1 3 @F @F @F @F

@END_Dcl

@END_Export

@BEG_Body
@TL(9)

(**************************************** WARNING ********************************************
 *** The KEBA Kemro K2 System including software is not intended for safety control tasks! ***
 ***                       For further information see Comment tab!                        ***
 *********************************************************************************************)
fbRTC(EN := FALSE);
sTime := DATE_AND_TIME_TO_STRING(fbRTC.CDT); //e.g. DT#2015-08-18-12:03:15.970149
sTimeStamp := CONCAT(MID(sTime, 10,4), '_', MID(sTime, 2, 15), '-',  MID(sTime, 2, 18), '-', MID(sTime, 2, 21)); //yyyy-mm-dd_hh-mm-ss

@END_Body

@END_Contents
